(* CoDeSys 2.3.9.36 project: KVR_Mast.bak.pro *)
(* Version: 01 *)
(* Author: JB *)
(* Libraries: ifm_CR0401\ifm_CR0401_V030100.lib*30.7.20 10:49:34, ifm_RAWCan\ifm_RAWCan_NT_V020004.lib*27.10.21 18:23:48, ifm_CANopen\ifm_CANopen_NT_V020004.lib*27.10.21 18:23:48, ifm_CANopen\3S_CanDrv.lib*27.10.21 18:23:48, ifm_CANopen\3S_CANopenManager.lib*27.10.21 18:23:48, Util.lib 6.11.07 15:39:24, standard.lib 4.10.05 12:14:46, SysLibCallback.lib 26.9.08 17:43:52 *)

(* PLC configuration (modules and I/O channels)
Configuration [LocalConfiguration] node 0, in %IB0 out %QB0 {IFM_PARAM_WORD_TIME = 0}
Input/Output [LocalInputOutput] node 1, in %IB0 out %QB0
IN00 AT %IB0 [ChInputBool] Input 00 Bit
IN01 AT %IB1 [ChInputBool] Input 01 Bit
IN02 AT %IB2 [ChInputBool] Input 02 Bit
IN03 AT %IB3 [ChInputBool] Input 03 Bit
IN04 AT %IB4 [ChInputBool] Input 04 Bit
IN05 AT %IB5 [ChInputBool] Input 05 Bit
IN06 AT %IB6 [ChInputBool] Input 06 Bit
IN07 AT %IB7 [ChInputBool] Input 07 Bit
IN08 AT %IB8 [ChInputBool] Input 08 Bit
IN09 AT %IB9 [ChInputBool] Input 09 Bit
IN10 AT %IB10 [ChInputBool] Input 10 Bit
IN11 AT %IB11 [ChInputBool] Input 11 Bit
OUT00 AT %QB0 [ChOutputBool] Output 00 Bit
OUT01 AT %QB1 [ChOutputBool] Output 01 Bit
OUT02 AT %QB2 [ChOutputBool] Output 02 Bit
OUT03 AT %QB3 [ChOutputBool] Output 03 Bit
OUT04 AT %QB4 [ChOutputBool] Output 04 Bit
OUT05 AT %QB5 [ChOutputBool] Output 05 Bit
OUT06 AT %QB6 [ChOutputBool] Output 06 Bit
OUT07 AT %QB7 [ChOutputBool] Output 07 Bit
System Inputs [LocalSystemInputs] node 2, in %IB12 out %QB8
  SUPPLY_VOLTAGE_VBBS AT %IW6 [ChInputWord] Supply voltage VBBS
  SUPPLY_VOLTAGE_VU AT %IW7 [ChInputWord] Supply voltage VU
  SUPPLY_VOLTAGE_VBB1 AT %IW8 [ChInputWord] Supply voltage VBB1
  SUPPLY_VOLTAGE_VBB2 AT %IW9 [ChInputWord] Supply voltage VBB2
  TEMPERATURE AT %IW10 [ChInputInt] Temperature
J1939 Interface [CAN_J1939] node 1, in %IB44 out %QB16
J1939 Interface [CAN_J1939] node 1, in %IB44 out %QB16
*)

(* Global variable list: Global_Constants *)
VAR_GLOBAL CONSTANT

	MAX_CTRLINDEX: BYTE := 0;

	SIMULATIONSMODUS: BOOL := FALSE;

	(* Flag positions for variable FlagsECU2PC *)
	ECU2PC_AllowRemote: INT := 3;
	ECU2PC_EmergencyStop: INT := 4;
	ECU2PC_RemoteAckn: INT := 6;
	ECU2PC_MainSwitch: INT := 7;

	(* Flag positions for variable FlagsPC2ECU *)
	PC2ECU_Remote: INT := 0;
	PC2ECU_BlackOut: INT := 1;
	PC2ECU_ResetMotorActiveTime: INT := 3;

	(* Flag positions for variables Mast[x].FlagsECU2PC *)
	ECU2PC_TopPosition: INT := 0;
	ECU2PC_BottomPosition: INT := 1;
	ECU2PC_MovingUp: INT := 2;
	ECU2PC_MovingDown: INT := 3;
	ECU2PC_LocalUp: INT := 4;
	ECU2PC_LocalDown: INT := 5;
	ECU2PC_LimitSwitch4m: INT := 7;
	ECU2PC_LimitSwitchBottom: INT := 8;
	ECU2PC_NotReadyToSwitchOn: INT := 9;
	ECU2PC_ParkPosition: INT := 10;
	ECU2PC_MontagePos: INT := 11;

	(* Flag positions for variables Mast[x].FlagsPC2ECU *)
	PC2ECU_MoveUp: INT := 0;
	PC2ECU_MoveDown: INT := 1;
	PC2ECU_SlowSpeed: INT := 2;

	(* Flag positions for variable Mast[x].ErrorECU2PC *)
	ECU2PC_ErrorFU: INT 					:= 0;
	ECU2PC_ErrorCanTimeout: INT 			:= 1;
	ECU2PC_ErrorFUPos: INT 					:= 6;
	ECU2PC_ErrorEndschalterUnten1: INT 		:= 7;
	ECU2PC_ErrorEndschalterUnten2: INT 		:= 8;
	ECU2PC_ErrorCurrentLimit: INT			:= 9;
	ECU2PC_ErrorSetMastHeight: INT			:= 10;

	QSCMD_NOP: BYTE				:= 0;
	QSCMD_CLEAR_ERROR: BYTE		:= 1;
	QSCMD_QUICK_STOP: BYTE		:= 113;
	QSCMD_HALT: BYTE			:= 114;
	QSCMD_VELOCITY_MODE: BYTE	:= 117; (* QSData0 = desired velocity *)
	QSCMD_ABS_POS_MODE: BYTE	:= 118; (* QSData0 = desired velocity, QSData1 = desired position *)

	(* Flag positions for FU statusword *)
	STAT_ENABLED: INT			:= 0;
	STAT_ERROR: INT				:= 1;
	STAT_WARNING: INT			:= 2;
	STAT_MOVING: INT			:= 3;
	STAT_REACHED: INT			:= 4;
	STAT_LIMIT: INT				:= 5;
	STAT_STOP_OR_HALT: INT		:= 11;

	FU1_POS_TO_MM: REAL 		:= 3.2573E-004;

	CAN_CHANNEL_HOST: BYTE 		:= 2;
	CAN_CHANNEL_LOCAL: BYTE 	:= 1;

	FU1_NODE_ID: BYTE			:= 127;

END_VAR

(* Global variable list: Global_Variables *)
VAR_GLOBAL

	BlinkSlow: BOOL;

	MasterPresent: BOOL;

	inputs: TYPE_INPUTS;
	outputs: TYPE_OUTPUTS;

	canNodeFU1Present: BOOL;

	tasteAuf: BOOL;
	tasteAb: BOOL;

	FlagsECU2PC: WORD			{parameter list=proc_vars_ecu [name=FlagsECU2PC 					index=16#3000 subindex=1 accessright="read only"] };
	FlagsPC2ECU: WORD			{parameter list=proc_vars_ecu [name=FlagsPC2ECU 					index=16#3000 subindex=2 accessright="write only"] };
	Windspeed: BYTE				{parameter list=proc_vars_ecu [name=Windspeed	 					index=16#3000 subindex=3 accessright="read only"] };
	CabinetTemperature: SINT	{parameter list=proc_vars_ecu [name=Temperature	 					index=16#3000 subindex=4 accessright="read only"] };
	ExtTemperature: SINT		{parameter list=proc_vars_ecu [name=ExtTemperature	 				index=16#3000 subindex=5 accessright="read only"] };
	IntVoltage: WORD			{parameter list=proc_vars_ecu [name=IntVoltage		 				index=16#3000 subindex=6 accessright="read only"] };

	Mast1Height: WORD			{parameter list=proc_vars_mast1 [name=Mast1Height 					index=16#3001 subindex=1 accessright="read only"] };
	Mast1FlagsECU2PC: WORD		{parameter list=proc_vars_mast1 [name=Mast1FlagsECU2PC 				index=16#3003 subindex=1 accessright="read only"] };
	Mast1FlagsPC2ECU: WORD		{parameter list=proc_vars_mast1 [name=Mast1FlagsPC2ECU 				index=16#3004 subindex=1 accessright="write only"] };
	Mast1Current: DINT			{parameter list=proc_vars_mast1 [name=Mast1Current 					index=16#3006 subindex=1 accessright="read only"] };
	Mast1ErrorECU2PC: WORD		{parameter list=proc_vars_mast1 [name=Mast1ErrorECU2PC				index=16#300D subindex=1 accessright="read only"] };
	Mast1FUErrorCode: WORD		{parameter list=proc_vars_mast1 [name=Mast1FUErrorCode				index=16#3010 subindex=1 accessright="read only"] };
	Mast1Speed: DINT			{parameter list=proc_vars_mast1 [name=Mast1Speed					index=16#3013 subindex=1 accessright="read only"] };

	(*
	Mast1TempPcbPower: WORD		{parameter list=proc_vars_mast1 [name=Mast1TempPcbPower				index=16#300A subindex=1 accessright="read only"] };
	Mast1TempPcbController: WORD{parameter list=proc_vars_mast1 [name=Mast1TempPcbController		index=16#300B subindex=1 accessright="read only"] };
	Mast1TempPcbAmplifier: WORD	{parameter list=proc_vars_mast1 [name=Mast1TempPcbAmplifier			index=16#300F subindex=1 accessright="read only"] };
	*)

	Mast1SetEncoderPW: DWORD	{parameter list=Parameters 		[name=Mast1SetEncoderPW				index=16#2014 subindex=1 accessright="read-write"] };

	Version: BYTE				{parameter list=version_info 	[name=Version						index=16#3020 subindex=1 accessright="read only"] };
	VersionDate: DWORD			{parameter list=version_info 	[name=VersionDate					index=16#3020 subindex=2 accessright="read only"] };

	Mast1MotorActiveTimeSeconds2: DWORD {parameter list=proc_vars_mast1 [name=Mast1MotorActiveTimeSeconds2 index=16#3014 subindex=1 accessright="read only"] };

	FU1_Current_Sim: DINT;

END_VAR

(* Global variable list: Parameters *)
VAR_GLOBAL RETAIN
	SettingsPW: DWORD := 0	 					{parameter list=Parameters [name=SettingsPW					 	index=16#2000 subindex=12 accessright="read-write"] };
	Mast1TopPosition: WORD := 9000 				{parameter list=Parameters [name=Mast1TopPosition 				index=16#2006 subindex=1 accessright="read-write"] };
	Mast1BottomPosition: WORD := 1675			{parameter list=Parameters [name=Mast1BottomPosition			index=16#2007 subindex=1 accessright="read-write"] };
	Mast1VelocityNormal: INT := 2500			{parameter list=Parameters [name=Mast1VelocityNormal			index=16#200A subindex=1 accessright="read-write"] };
	Mast1VelocityBottom: INT := 500				{parameter list=Parameters [name=Mast1VelocityBottom			index=16#200C subindex=1 accessright="read-write"] };
	Mast1BottomPositionOffset: WORD := 130		{parameter list=Parameters [name=Mast1BottomPositionOffset		index=16#200D subindex=1 accessright="read-write"] };
	Mast1CurrentLimitBottom: INT := 30			{parameter list=Parameters [name=Mast1CurrentLimitBottom		index=16#200E subindex=1 accessright="read-write"] };
	Mast1BottomLimitSwitchWindow: WORD := 100	{parameter list=Parameters [name=Mast1BottomLimitSwitchWindow	index=16#200F subindex=1 accessright="read-write"] };
	Mast1MontagePos: WORD := 2000 				{parameter list=Parameters [name=Mast1MontagePos 				index=16#2010 subindex=1 accessright="read-write"] };
	Mast1MotorActiveTimeSeconds: DWORD := 0		{parameter list=Parameters [name=Mast1MotorActiveTimeSeconds	index=16#2013 subindex=1 accessright="read-write"] };
	Mast1CurrentLimit: INT := 40				{parameter list=Parameters [name=Mast1CurrentLimit				index=16#2018 subindex=1 accessright="read-write"] };
	Mast1TopSettlingOffset: INT := 40			{parameter list=Parameters [name=Mast1TopSettlingOffset			index=16#2019 subindex=1 accessright="read-write"] };
END_VAR

(* Data type *)
TYPE TYPE_INPUTS :
	STRUCT
		TasteAusfahren: BOOL;
		TasteEinfahren: BOOL;
		TastePoweredByGenerator: BOOL;
		EndschalterNotantrieb: BOOL;
		EndschalterEingefahren: BOOL;
		EndschalterAufgerichtet: BOOL;
	END_STRUCT
END_TYPE

(* Data type *)
TYPE TYPE_OUTPUTS :
	STRUCT
		LEDAusgefahren: BOOL;
		LEDEingefahren: BOOL;
		LEDMontagePos: BOOL;
		RelaisMotorLeistung: BOOL;
		SchuetzGrundlast: BOOL;
	END_STRUCT
END_TYPE

(* POU PLC_PRG, FBD *)
PROGRAM PLC_PRG
VAR
	Init1: BOOL:=TRUE;
	CycleTime:DWORD;
	MaxCycleTime:DWORD;
	ResetMax:BOOL;
END_VAR
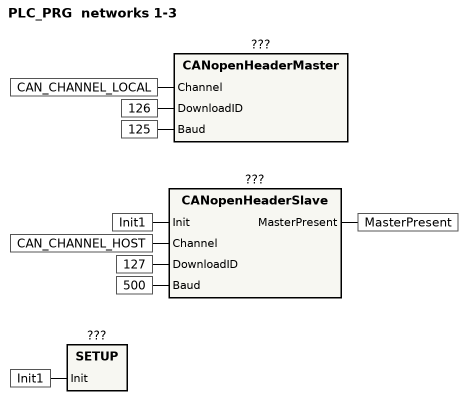
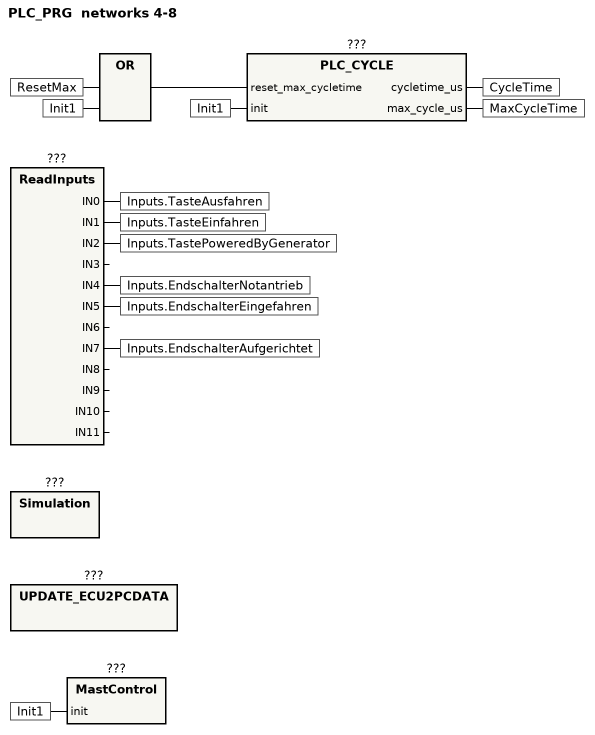
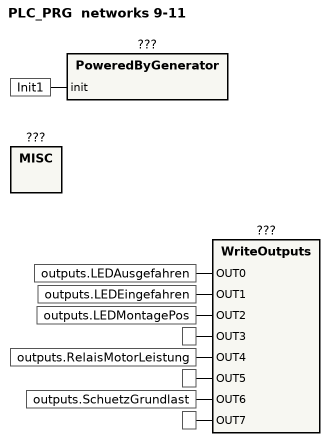
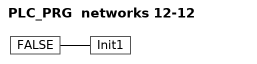
_FBD_ (* Function Block Diagram *)
NETWORK 1 (* CAN Master auf CAN1 initialisieren (Schnittstelle zu FU) *)
	???:CANopenHeaderMaster(Channel: CAN_CHANNEL_LOCAL, DownloadID: 126, Baud: 125)
NETWORK 2 (* CAN Slave auf CAN2 initialisieren (Schnittstelle zu PC) *)
	???:CANopenHeaderSlave(Init: Init1, Channel: CAN_CHANNEL_HOST, DownloadID: 127, Baud: 500) => MasterPresent
NETWORK 3
	???:SETUP(Init: Init1)
NETWORK 4
	???:PLC_CYCLE(reset_max_cycletime: OR(ResetMax, Init1), init: Init1, max_cycle_us => MaxCycleTime) => CycleTime
NETWORK 5
	???:ReadInputs(IN1 => Inputs.TasteEinfahren, IN2 => Inputs.TastePoweredByGenerator, IN4 => Inputs.EndschalterNotantrieb, IN5 => Inputs.EndschalterEingefahren, IN7 => Inputs.EndschalterAufgerichtet) => Inputs.TasteAusfahren
NETWORK 6
	???:Simulation()
NETWORK 7
	???:UPDATE_ECU2PCDATA()
NETWORK 8
	NOT ???:MastControl(init: Init1)
NETWORK 9
	???:PoweredByGenerator(init: Init1)
NETWORK 10
	???:MISC()
NETWORK 11
	???:WriteOutputs(OUT0: outputs.LEDAusgefahren, OUT1: outputs.LEDEingefahren, OUT2: outputs.LEDMontagePos, OUT3: , OUT4: outputs.RelaisMotorLeistung, OUT5: , OUT6: outputs.SchuetzGrundlast, OUT7: )
NETWORK 12 (* last line *)
	FALSE => Init1
_END_FBD_
(* the same logic as Structured Text *)
(* Network 1: see the listing above *)
(* Network 2: see the listing above *)
(* Network 3: see the listing above *)
(* Network 4: see the listing above *)
(* Network 5: see the listing above *)
(* Network 6: see the listing above *)
(* Network 7: see the listing above *)
(* Network 8: see the listing above *)
(* Network 9: see the listing above *)
(* Network 10: see the listing above *)
(* Network 11: see the listing above *)
(* Network 12 *)
Init1 := FALSE;
END_PROGRAM

(* POU CANopen/CANopenHeaderMaster, FBD *)
PROGRAM CANopenHeaderMaster
VAR_INPUT
	Channel: BYTE;
	DownloadID: BYTE;
	Baud: WORD;
END_VAR
VAR
	(*CAN settings*)
	SettingsCAN: CAN_SETTING_ST;

	(*Set CANopen state*)
	SetCanOpenState: CANOPEN_SETSTATE;
	SetState:BOOL:=TRUE;

	(*Handling CANopen status*)
	HandlingCANopen: CANopen_HANDLING_ST;
	Baudrate: DWORD;
	MasterState: BYTE;
	GuardError: BOOL;
	ErrorNodeList: ARRAY[0..MAXGUARDERR] OF BYTE;
	CanState: BYTE;
	Nodestate: BYTE;
	LastNodeState: BYTE;

	(*Emergency handling*)
	CanEmcy: CAN_EMCY;
	RestEmcyList: BOOL;
	EMCY_MSG_Count: DWORD; (* No of EMCY messages  Leaving errors are count too *)
	EmcyStruct: ARRAY[0..10] OF tT_EMCY;

	(*Handling CAN status*)
	StatusCan: CAN_Status_and_Errors;
	ResetCanFlags: BOOL;
	BusLoad: BYTE;
	BusOff: BOOL;
	RxOverflow: BOOL;
	RxWarning: BOOL;
	TxOverflow: BOOL;
	TxWarning: BOOL;

	GetstateSlave1: CANopen_GetStateSlave;

END_VAR
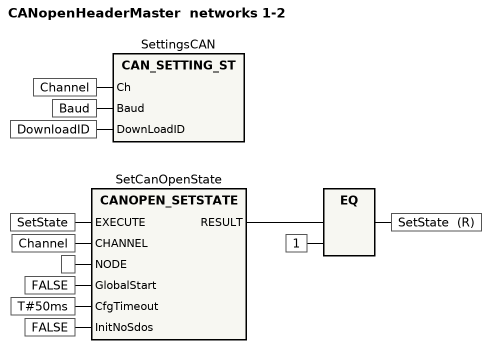
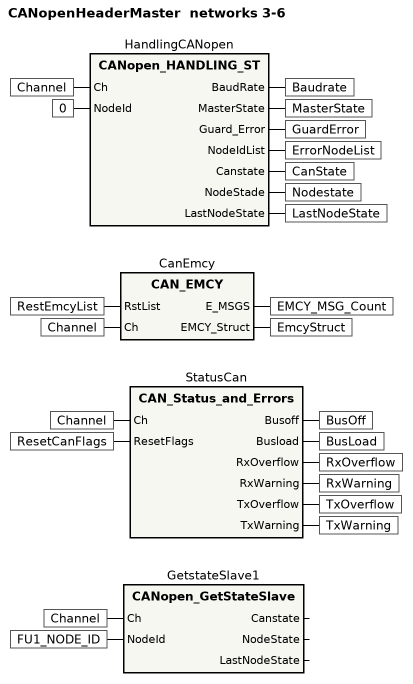
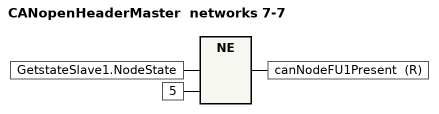
_FBD_ (* Function Block Diagram *)
NETWORK 1 (* Basic functions for the CAN / CANopen functionality *)
	SettingsCAN:CAN_SETTING_ST(Ch: Channel, Baud: Baud, DownLoadID: DownloadID)
NETWORK 2 (* Set CANopen status *)
	EQ(SetCanOpenState:CANOPEN_SETSTATE(EXECUTE: SetState, CHANNEL: Channel, NODE: , GlobalStart: FALSE, CfgTimeout: T#50ms, InitNoSdos: FALSE), 1) => R SetState
NETWORK 3 (* CANopen Master and heartbeat handling *)
	HandlingCANopen:CANopen_HANDLING_ST(Ch: Channel, NodeId: 0, MasterState => MasterState, Guard_Error => GuardError, NodeIdList => ErrorNodeList, Canstate => CanState, NodeStade => Nodestate, LastNodeState => LastNodeState) => Baudrate
NETWORK 4 (* CANopen Emergency Handling for 11 emergency messages *)
	CanEmcy:CAN_EMCY(RstList: RestEmcyList, Ch: Channel, EMCY_Struct => EmcyStruct) => EMCY_MSG_Count
NETWORK 5 (* Get the CAN Status and CAN Errors *)
	StatusCan:CAN_Status_and_Errors(Ch: Channel, ResetFlags: ResetCanFlags, Busload => BusLoad, RxOverflow => RxOverflow, RxWarning => RxWarning, TxOverflow => TxOverflow, TxWarning => TxWarning) => BusOff
NETWORK 6
	GetstateSlave1:CANopen_GetStateSlave(Ch: Channel, NodeId: FU1_NODE_ID)
NETWORK 7
	NE(GetstateSlave1.NodeState, 5) => R canNodeFU1Present
_END_FBD_
(* the same logic as Structured Text *)
(* Network 1 *)
SettingsCAN(Ch := Channel, Baud := Baud, DownLoadID := DownloadID);
(* Network 2: see the listing above *)
(* Network 3 *)
HandlingCANopen(Ch := Channel, NodeId := 0);
MasterState := HandlingCANopen.MasterState;
GuardError := HandlingCANopen.Guard_Error;
ErrorNodeList := HandlingCANopen.NodeIdList;
CanState := HandlingCANopen.Canstate;
Nodestate := HandlingCANopen.NodeStade;
LastNodeState := HandlingCANopen.LastNodeState;
Baudrate := HandlingCANopen.BaudRate;
(* Network 4 *)
CanEmcy(RstList := RestEmcyList, Ch := Channel);
EmcyStruct := CanEmcy.EMCY_Struct;
EMCY_MSG_Count := CanEmcy.E_MSGS;
(* Network 5 *)
StatusCan(Ch := Channel, ResetFlags := ResetCanFlags);
BusLoad := StatusCan.Busload;
RxOverflow := StatusCan.RxOverflow;
RxWarning := StatusCan.RxWarning;
TxOverflow := StatusCan.TxOverflow;
TxWarning := StatusCan.TxWarning;
BusOff := StatusCan.Busoff;
(* Network 6 *)
GetstateSlave1(Ch := Channel, NodeId := FU1_NODE_ID);
(* Network 7 *)
IF GetstateSlave1.NodeState <> 5 THEN canNodeFU1Present := FALSE; END_IF;
END_PROGRAM

(* POU CANopen/CAN_SETTING_ST, ST *)
FUNCTION_BLOCK CAN_SETTING_ST
(* Basic functions for the CAN / CANopen functionality *)
VAR

	CAN_SETDOWNLOADID_: CAN_SETDOWNLOADID;
	CAN_ENABLE_: CAN_ENABLE;
	CANOPEN_ENABLE_: CANOPEN_ENABLE;

	CANOPEN_SETSTATE_: CANOPEN_SETSTATE;
END_VAR
VAR_INPUT
	Ch: BYTE;
	Baud:WORD;
	DownLoadID:BYTE;
END_VAR
CAN_SETDOWNLOADID_(EXECUTE:=TRUE , CHANNEL:=Ch , DOWNLOAD_ID:=DownLoadID , RESULT=> );
CAN_ENABLE_(ENABLE:=TRUE , CHANNEL:=Ch , BAUDRATE:=Baud , RESULT=> );
CANOPEN_ENABLE_(ENABLE:=TRUE , CHANNEL:=Ch , Baudrate:=Baud , RESULT=> );
END_FUNCTION_BLOCK

(* POU CANopen/CANopen_HANDLING_ST, ST *)
FUNCTION_BLOCK CANopen_HANDLING_ST
(* CANopen Master and heartbeat handling *)
VAR
	CANOPEN_GETSTATE_: CANOPEN_GETSTATE;
	Execute_Getstate: BOOL := TRUE;
	CANOPEN_GETGUARDHBERRLIST_: CANOPEN_GETGUARDHBERRLIST;
	Execute_Guardlst: BOOL := TRUE;
	ResetErrorList: BOOL;
	PlcNodeId: BYTE;
	i: INT;
	GuardErrorCnt: WORD;
END_VAR
VAR_INPUT
	Ch: BYTE;
	NodeId: BYTE;
END_VAR
VAR_OUTPUT
	BaudRate: DWORD;
	MasterState: BYTE;
	Guard_Error: BOOL;
	NodeIdList: ARRAY[0..MAXGUARDERR] OF BYTE;
	Canstate: BYTE;
	NodeStade: BYTE;
	LastNodeState: BYTE;
END_VAR
(* ^^^^ Get the current state of the CANopen master ^^^^ *)
CANOPEN_GETSTATE_(
	EXECUTE:=Execute_Getstate ,
	CHANNEL:=Ch ,
	NODE:=NodeId ,
	MASTERSTATE=>MasterState ,
	PLCNODEID=>PlcNodeId ,
	PLCBAUDRATE=>BaudRate ,
	PLCVERSION=>,
	CANSTATE=>Canstate ,
	NODESTATE=>NodeStade ,
	LASTNODESTATE=>LastNodeState ,
	RESULT=> );

(* Values are valid now, function call can be stopped *)
IF CANOPEN_GETSTATE_.RESULT= 1 THEN
	Execute_Getstate:=FALSE;
END_IF

(* Function is passive, execute again *)
IF CANOPEN_GETSTATE_.RESULT= 0 THEN
	Execute_Getstate:=TRUE;
END_IF

(* ^^^^^ Get heartbeaterror or nodeguarding error ^^^^ *)
CANOPEN_GETGUARDHBERRLIST_(
	EXECUTE:=Execute_Guardlst ,
	CHANNEL:=Ch ,
	ResetList:=ResetErrorList ,
	N_NODES=>GuardErrorCnt,
	NODEID=>NodeIdList ,
	RESULT=> );

(* Values are valid now, function call can be stopped *)
IF CANOPEN_GETGUARDHBERRLIST_.RESULT= 1 THEN
	Execute_Guardlst:= FALSE;
END_IF

(* Function is passive, execute again *)
IF CANOPEN_GETGUARDHBERRLIST_.RESULT= 0 THEN
	Execute_Guardlst:= TRUE;
END_IF

(* An heartbeaterror has been appeared *)
IF CANOPEN_GETGUARDHBERRLIST_.N_NODES >0 THEN
	Guard_Error:=TRUE;
ELSE
	Guard_Error:=FALSE;
END_IF;

IF Ch = CAN_CHANNEL_LOCAL THEN

	canNodeFU1Present := TRUE;
	
	FOR i := 0 TO GuardErrorCnt DO
		IF FU1_NODE_ID = NodeIdList[i] THEN
			canNodeFU1Present := FALSE;
		END_IF
	END_FOR

END_IF
END_FUNCTION_BLOCK

(* POU CANopen/CAN_EMCY, FBD *)
FUNCTION_BLOCK CAN_EMCY
VAR_INPUT
	RstList: BOOL;
	Ch: BYTE;
END_VAR
VAR_OUTPUT
	E_MSGS: DWORD;
	EMCY_Struct: ARRAY[0..10] OF tT_EMCY;
END_VAR
VAR
	CANOPEN_GETEMCYMESSAGES_: CANOPEN_GETEMCYMESSAGES;
	Get_EMCY_MSG: BOOL := TRUE;
END_VAR
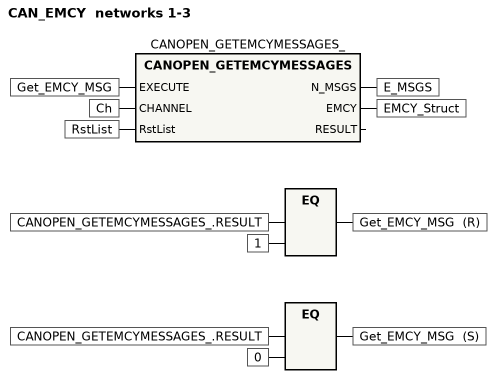
_FBD_ (* Function Block Diagram *)
NETWORK 1
	CANOPEN_GETEMCYMESSAGES_:CANOPEN_GETEMCYMESSAGES(EXECUTE: Get_EMCY_MSG, CHANNEL: Ch, RstList: RstList, EMCY => EMCY_Struct) => E_MSGS
NETWORK 2
	EQ(CANOPEN_GETEMCYMESSAGES_.RESULT, 1) => R Get_EMCY_MSG
NETWORK 3
	EQ(CANOPEN_GETEMCYMESSAGES_.RESULT, 0) => S Get_EMCY_MSG
_END_FBD_
(* the same logic as Structured Text *)
(* Network 1 *)
CANOPEN_GETEMCYMESSAGES_(EXECUTE := Get_EMCY_MSG, CHANNEL := Ch, RstList := RstList);
EMCY_Struct := CANOPEN_GETEMCYMESSAGES_.EMCY;
E_MSGS := CANOPEN_GETEMCYMESSAGES_.N_MSGS;
(* Network 2 *)
IF CANOPEN_GETEMCYMESSAGES_.RESULT = 1 THEN Get_EMCY_MSG := FALSE; END_IF;
(* Network 3 *)
IF CANOPEN_GETEMCYMESSAGES_.RESULT = 0 THEN Get_EMCY_MSG := TRUE; END_IF;
END_FUNCTION_BLOCK

(* POU CANopen/CAN_Status_and_Errors, FBD *)
FUNCTION_BLOCK CAN_Status_and_Errors
(* Get the CAN Status and CAN Errors *)
VAR

	CanStatus:CAN_STATUS;
	GETBUFFERFLAGS: CANOPEN_GETBUFFERFLAGS;

	ExecuteBufferFlags: BOOL:=TRUE;

END_VAR
VAR_INPUT
	Ch: BYTE;

	ResetFlags: BOOL;
END_VAR
VAR_OUTPUT
	Busoff: BOOL;
	Busload: BYTE;
	RxOverflow: BOOL;
	RxWarning: BOOL;
	TxOverflow: BOOL;
	TxWarning: BOOL;
END_VAR
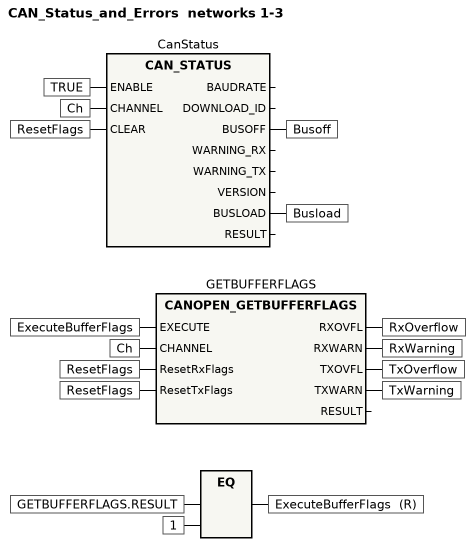
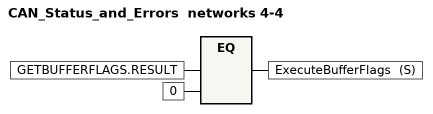
_FBD_ (* Function Block Diagram *)
NETWORK 1 (* Get the CAN Status *)
	CanStatus:CAN_STATUS(ENABLE: TRUE, CHANNEL: Ch, CLEAR: ResetFlags, BUSOFF => Busoff, BUSLOAD => Busload)
NETWORK 2 (* Get Buffer warnings / Reset Buffer Warning *)
	GETBUFFERFLAGS:CANOPEN_GETBUFFERFLAGS(EXECUTE: ExecuteBufferFlags, CHANNEL: Ch, ResetRxFlags: ResetFlags, ResetTxFlags: ResetFlags, RXWARN => RxWarning, TXOVFL => TxOverflow, TXWARN => TxWarning) => RxOverflow
NETWORK 3
	EQ(GETBUFFERFLAGS.RESULT, 1) => R ExecuteBufferFlags
NETWORK 4
	EQ(GETBUFFERFLAGS.RESULT, 0) => S ExecuteBufferFlags
_END_FBD_
(* the same logic as Structured Text *)
(* Network 1: Get the CAN Status *)
CanStatus(ENABLE := TRUE, CHANNEL := Ch, CLEAR := ResetFlags);
Busoff := CanStatus.BUSOFF;
Busload := CanStatus.BUSLOAD;
(* Network 2: Get Buffer warnings / Reset Buffer Warning *)
GETBUFFERFLAGS(EXECUTE := ExecuteBufferFlags, CHANNEL := Ch, ResetRxFlags := ResetFlags, ResetTxFlags := ResetFlags);
RxWarning := GETBUFFERFLAGS.RXWARN;
TxOverflow := GETBUFFERFLAGS.TXOVFL;
TxWarning := GETBUFFERFLAGS.TXWARN;
RxOverflow := GETBUFFERFLAGS.RXOVFL;
(* Network 3 *)
IF GETBUFFERFLAGS.RESULT = 1 THEN ExecuteBufferFlags := FALSE; END_IF;
(* Network 4 *)
IF GETBUFFERFLAGS.RESULT = 0 THEN ExecuteBufferFlags := TRUE; END_IF;
END_FUNCTION_BLOCK

(* POU CANopen/CANopen_GetStateSlave, ST *)
FUNCTION_BLOCK CANopen_GetStateSlave
VAR
	CANOPEN_GETSTATE_: CANOPEN_GETSTATE;
	Execute_Getstate: BOOL := TRUE;
END_VAR
VAR_INPUT
	Ch: BYTE;
	NodeId: BYTE;
END_VAR
VAR_OUTPUT
	Canstate: BYTE;
	NodeState: BYTE;
	LastNodeState: BYTE;
END_VAR
CANOPEN_GETSTATE_(
	EXECUTE:=Execute_Getstate ,
	CHANNEL:=Ch ,
	NODE:=NodeId ,
	MASTERSTATE=>,
	PLCNODEID=> ,
	PLCBAUDRATE=> ,
	PLCVERSION=>,
	CANSTATE=>Canstate ,
	NODESTATE=>NodeState ,
	LASTNODESTATE=>LastNodeState ,
	RESULT=> );

(* Values are valid now, function call can be stopped *)
IF CANOPEN_GETSTATE_.RESULT= 1 THEN
	Execute_Getstate:=FALSE;
END_IF

(* Function is passive, execute again *)
IF CANOPEN_GETSTATE_.RESULT= 0 THEN
	Execute_Getstate:=TRUE;
END_IF
END_FUNCTION_BLOCK

(* POU CANopen/CANopenHeaderSlave, FBD *)
PROGRAM CANopenHeaderSlave
VAR_INPUT
	Init: BOOL;
	Channel: BYTE;
	DownloadID: BYTE;
	Baud: WORD;
END_VAR
VAR_OUTPUT
	MasterPresent: BOOL;
END_VAR
VAR
	(*SettingsCAN*)
	SettingsCAN: CAN_SETTING_ST;

	(*Get status*)
	GetStateSlave: CANOPEN_GETNMTSTATESLAVE;
	SetGetStateSlave: BOOL;
	ResultState: BYTE;
	NodeState: BYTE;

	(*Get CANopen Node ID*)
	GetState: CANOPEN_GETSTATE;
	NodeId: BYTE;

	(*Get Guarding status*)
	GetGuard: CANOPEN_GETGUARDHBSTATSLV;
	GetGuardEx: BOOL;
	ResetGuard: BOOL;

END_VAR
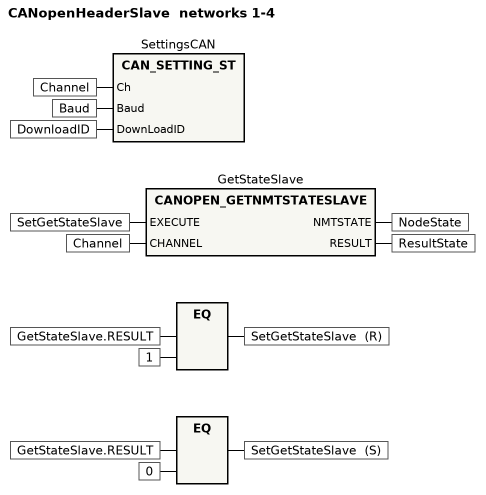
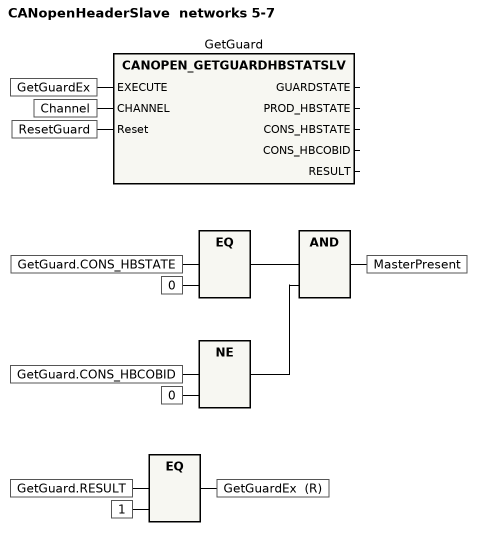
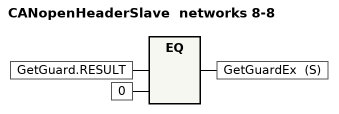
_FBD_ (* Function Block Diagram *)
NETWORK 1 (* Basic functions for the CAN / CANopen functionality *)
	SettingsCAN:CAN_SETTING_ST(Ch: Channel, Baud: Baud, DownLoadID: DownloadID)
NETWORK 2
	GetStateSlave:CANOPEN_GETNMTSTATESLAVE(EXECUTE: SetGetStateSlave, CHANNEL: Channel, RESULT => ResultState) => NodeState
NETWORK 3
	EQ(GetStateSlave.RESULT, 1) => R SetGetStateSlave
NETWORK 4
	EQ(GetStateSlave.RESULT, 0) => S SetGetStateSlave
NETWORK 5
	GetGuard:CANOPEN_GETGUARDHBSTATSLV(EXECUTE: GetGuardEx, CHANNEL: Channel, Reset: ResetGuard)
NETWORK 6
	AND(EQ(GetGuard.CONS_HBSTATE, 0), NE(GetGuard.CONS_HBCOBID, 0)) => MasterPresent
NETWORK 7
	EQ(GetGuard.RESULT, 1) => R GetGuardEx
NETWORK 8
	EQ(GetGuard.RESULT, 0) => S GetGuardEx
_END_FBD_
(* the same logic as Structured Text *)
(* Network 1: Basic functions for the CAN / CANopen functionality *)
SettingsCAN(Ch := Channel, Baud := Baud, DownLoadID := DownloadID);
(* Network 2 *)
GetStateSlave(EXECUTE := SetGetStateSlave, CHANNEL := Channel);
ResultState := GetStateSlave.RESULT;
NodeState := GetStateSlave.NMTSTATE;
(* Network 3 *)
IF GetStateSlave.RESULT = 1 THEN SetGetStateSlave := FALSE; END_IF;
(* Network 4 *)
IF GetStateSlave.RESULT = 0 THEN SetGetStateSlave := TRUE; END_IF;
(* Network 5 *)
GetGuard(EXECUTE := GetGuardEx, CHANNEL := Channel, Reset := ResetGuard);
(* Network 6 *)
MasterPresent := (GetGuard.CONS_HBSTATE = 0) AND (GetGuard.CONS_HBCOBID <> 0);
(* Network 7 *)
IF GetGuard.RESULT = 1 THEN GetGuardEx := FALSE; END_IF;
(* Network 8 *)
IF GetGuard.RESULT = 0 THEN GetGuardEx := TRUE; END_IF;
END_PROGRAM

(* POU Steuerung/SETUP, ST *)
PROGRAM SETUP
VAR_INPUT
	Init: BOOL;
END_VAR
VAR
	getAppInfo: GET_APP_INFO;
END_VAR
IF NOT Init THEN
	RETURN;
END_IF;

Mast1FlagsECU2PC.ECU2PC_ParkPosition := FALSE;

getAppInfo(ENABLE := TRUE);

VersionDate := STRING_TO_DWORD(LEFT(getAppInfo.BUILD_DATE, 8));
Version := STRING_TO_BYTE(LEFT(getAppInfo.VERSION, 3));
END_PROGRAM

(* POU PLC_CYCLE, ST *)
PROGRAM PLC_CYCLE
VAR_INPUT
	reset_max_cycletime: BOOL;
	init: BOOL;
END_VAR
VAR_OUTPUT
	cycletime_us: DWORD;
	max_cycle_us: DWORD;
END_VAR
VAR
	old_cycle: DWORD;
	TIMER_READ_US1: TIMER_READ_US;
	cycle: DWORD;
	nextTS: DWORD;
END_VAR
TIMER_READ_US1(TIME_US=>cycle );
cycletime_us:=cycle-old_cycle;
old_cycle:=cycle;

IF max_cycle_us<cycletime_us AND NOT init THEN
	max_cycle_us:=cycletime_us;
END_IF

IF reset_max_cycletime THEN
	max_cycle_us:=0;
END_IF

IF init THEN
	nextTS := cycle;
END_IF
(* Mehr als 1 Mio Ticks vergangen? *)
(* Zweikomplementarithmetik, d.h. funktioniert auch bei DWORD-Überlauf *)
IF cycle - nextTS > 1000000 THEN
	(* Das nächste Mal wieder nach 1 Mio Ticks (=1 Sekunde) *)
	nextTS := nextTS + 1000000;
	IF FU1_QSCmd <> QSCMD_HALT THEN
		Mast1MotorActiveTimeSeconds := Mast1MotorActiveTimeSeconds + 1;
	END_IF
END_IF
IF FlagsPC2ECU.PC2ECU_ResetMotorActiveTime THEN
	Mast1MotorActiveTimeSeconds := 0;
END_IF
END_PROGRAM

(* POU InputsOutputs/ReadInputs, FBD *)
PROGRAM ReadInputs
VAR
	_input: ARRAY[0..11] OF INPUT;
END_VAR
VAR_OUTPUT
	IN0: BOOL;
	IN1: BOOL;
	IN2: BOOL;
	IN3: BOOL;
	IN4: BOOL;
	IN5: BOOL;
	IN6: BOOL;
	IN7: BOOL;
	IN8: BOOL;
	IN9: BOOL;
	IN10: BOOL;
	IN11: BOOL;
END_VAR
VAR CONSTANT
	ModeInput_Off: BYTE := 0;
	ModeInput_0_10V: BYTE := 3;
	ModeInput_Ratio: BYTE := 6;
	ModeInput_0_20mA: BYTE := 7;
	ModeInput_0_32V: BYTE := 9;
	ModeInput_LowSide: BYTE := 10;
	ModeInput_LowSideNamur: BYTE := 11;
	ModeInput_HighSide: BYTE := 12;
	ModeInput_Resistor: BYTE := 18;
END_VAR
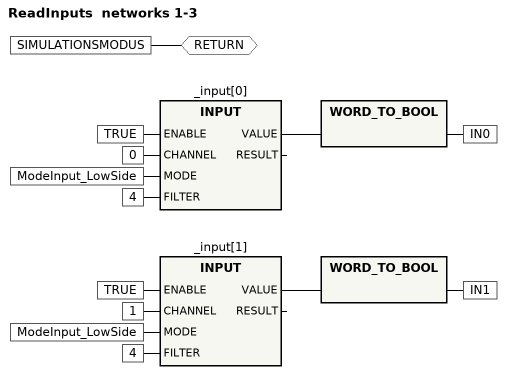
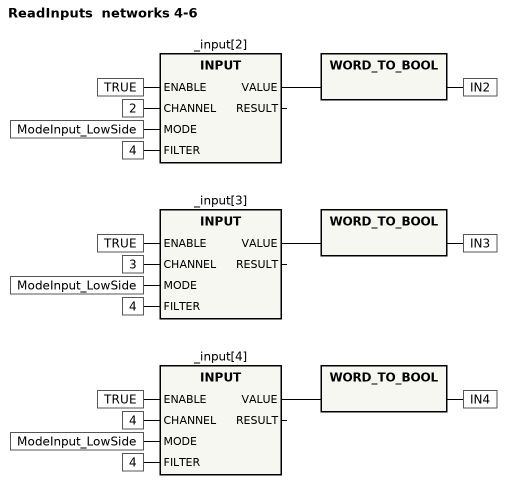
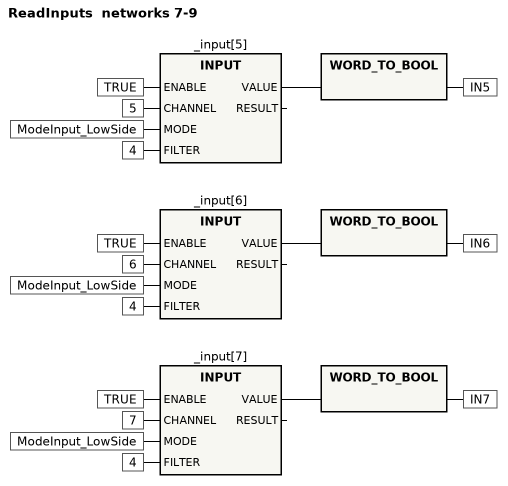
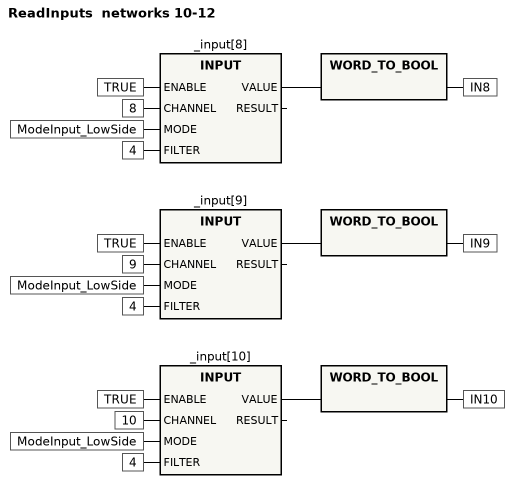
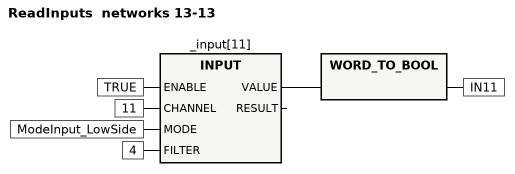
_FBD_ (* Function Block Diagram *)
NETWORK 1
	SIMULATIONSMODUS => <RETURN>
NETWORK 2
	WORD_TO_BOOL(_input[0]:INPUT(ENABLE: TRUE, CHANNEL: 0, MODE: ModeInput_LowSide, FILTER: 4)) => IN0
NETWORK 3
	WORD_TO_BOOL(_input[1]:INPUT(ENABLE: TRUE, CHANNEL: 1, MODE: ModeInput_LowSide, FILTER: 4)) => IN1
NETWORK 4
	WORD_TO_BOOL(_input[2]:INPUT(ENABLE: TRUE, CHANNEL: 2, MODE: ModeInput_LowSide, FILTER: 4)) => IN2
NETWORK 5
	WORD_TO_BOOL(_input[3]:INPUT(ENABLE: TRUE, CHANNEL: 3, MODE: ModeInput_LowSide, FILTER: 4)) => IN3
NETWORK 6
	WORD_TO_BOOL(_input[4]:INPUT(ENABLE: TRUE, CHANNEL: 4, MODE: ModeInput_LowSide, FILTER: 4)) => IN4
NETWORK 7
	WORD_TO_BOOL(_input[5]:INPUT(ENABLE: TRUE, CHANNEL: 5, MODE: ModeInput_LowSide, FILTER: 4)) => IN5
NETWORK 8
	WORD_TO_BOOL(_input[6]:INPUT(ENABLE: TRUE, CHANNEL: 6, MODE: ModeInput_LowSide, FILTER: 4)) => IN6
NETWORK 9
	WORD_TO_BOOL(_input[7]:INPUT(ENABLE: TRUE, CHANNEL: 7, MODE: ModeInput_LowSide, FILTER: 4)) => IN7
NETWORK 10
	WORD_TO_BOOL(_input[8]:INPUT(ENABLE: TRUE, CHANNEL: 8, MODE: ModeInput_LowSide, FILTER: 4)) => IN8
NETWORK 11
	WORD_TO_BOOL(_input[9]:INPUT(ENABLE: TRUE, CHANNEL: 9, MODE: ModeInput_LowSide, FILTER: 4)) => IN9
NETWORK 12
	WORD_TO_BOOL(_input[10]:INPUT(ENABLE: TRUE, CHANNEL: 10, MODE: ModeInput_LowSide, FILTER: 4)) => IN10
NETWORK 13
	WORD_TO_BOOL(_input[11]:INPUT(ENABLE: TRUE, CHANNEL: 11, MODE: ModeInput_LowSide, FILTER: 4)) => IN11
_END_FBD_
(* the same logic as Structured Text *)
(* Network 1 *)
IF SIMULATIONSMODUS THEN RETURN; END_IF;
(* Network 2 *)
_input[0](ENABLE := TRUE, CHANNEL := 0, MODE := ModeInput_LowSide, FILTER := 4);
IN0 := WORD_TO_BOOL(_input[0].VALUE);
(* Network 3 *)
_input[1](ENABLE := TRUE, CHANNEL := 1, MODE := ModeInput_LowSide, FILTER := 4);
IN1 := WORD_TO_BOOL(_input[1].VALUE);
(* Network 4 *)
_input[2](ENABLE := TRUE, CHANNEL := 2, MODE := ModeInput_LowSide, FILTER := 4);
IN2 := WORD_TO_BOOL(_input[2].VALUE);
(* Network 5 *)
_input[3](ENABLE := TRUE, CHANNEL := 3, MODE := ModeInput_LowSide, FILTER := 4);
IN3 := WORD_TO_BOOL(_input[3].VALUE);
(* Network 6 *)
_input[4](ENABLE := TRUE, CHANNEL := 4, MODE := ModeInput_LowSide, FILTER := 4);
IN4 := WORD_TO_BOOL(_input[4].VALUE);
(* Network 7 *)
_input[5](ENABLE := TRUE, CHANNEL := 5, MODE := ModeInput_LowSide, FILTER := 4);
IN5 := WORD_TO_BOOL(_input[5].VALUE);
(* Network 8 *)
_input[6](ENABLE := TRUE, CHANNEL := 6, MODE := ModeInput_LowSide, FILTER := 4);
IN6 := WORD_TO_BOOL(_input[6].VALUE);
(* Network 9 *)
_input[7](ENABLE := TRUE, CHANNEL := 7, MODE := ModeInput_LowSide, FILTER := 4);
IN7 := WORD_TO_BOOL(_input[7].VALUE);
(* Network 10 *)
_input[8](ENABLE := TRUE, CHANNEL := 8, MODE := ModeInput_LowSide, FILTER := 4);
IN8 := WORD_TO_BOOL(_input[8].VALUE);
(* Network 11 *)
_input[9](ENABLE := TRUE, CHANNEL := 9, MODE := ModeInput_LowSide, FILTER := 4);
IN9 := WORD_TO_BOOL(_input[9].VALUE);
(* Network 12 *)
_input[10](ENABLE := TRUE, CHANNEL := 10, MODE := ModeInput_LowSide, FILTER := 4);
IN10 := WORD_TO_BOOL(_input[10].VALUE);
(* Network 13 *)
_input[11](ENABLE := TRUE, CHANNEL := 11, MODE := ModeInput_LowSide, FILTER := 4);
IN11 := WORD_TO_BOOL(_input[11].VALUE);
END_PROGRAM

(* POU Steuerung/Simulation, ST *)
PROGRAM Simulation
VAR
	cnt: WORD;
END_VAR
IF NOT SIMULATIONSMODUS THEN
	RETURN;
END_IF

inputs.EndschalterEingefahren := Mast1Height <= Mast1BottomPosition+2;

IF Mast1Height < Mast1BottomPosition THEN
	Mast1Height := Mast1BottomPosition;
END_IF

FU1_Current_Sim := 0;

IF FU1_QSCmd = QSCMD_ABS_POS_MODE THEN
	IF MastControl.zielposition > Mast1Height THEN
		Mast1Height := Mast1Height + 1;
		FU1_Current_Sim := 10;
	END_IF
	IF MastControl.zielposition < Mast1Height THEN
		Mast1Height := Mast1Height - 1;
		FU1_Current_Sim := 10;
	END_IF
ELSIF FU1_QSCmd = QSCMD_VELOCITY_MODE THEN
	IF cnt > 0 THEN
		cnt := cnt - 1;
	ELSE
		cnt := 10;
		Mast1Height := Mast1Height - 1;
	END_IF
	IF Mast1Height = Mast1BottomPosition THEN
		FU1_Current_Sim := 35;
	ELSE
		FU1_Current_Sim := 10;
	END_IF
END_IF
END_PROGRAM

(* POU Steuerung/MastControl, ST *)
PROGRAM MastControl
VAR_INPUT
	init: BOOL;
END_VAR
VAR
	aufbauen: BOOL;
	abbauen: BOOL;
	zielposition: WORD := 1;
	rtTasteAuf: R_TRIG;
	rtTasteAb: R_TRIG;
	rtTasteReset: R_TRIG;
	rtMastEingefahren: R_TRIG;
	rtSystemEin: R_TRIG;
	resetMasthoehe: BOOL;
	masthoeheReal: REAL;
	FUValue: DWORD;
	SDOWriteOffset: CANOPEN_SDOWRITE;
	SDOData: ARRAY[0..3] OF BYTE;
	TSStart: DWORD;
	tonSystemEin: TON;
	tonKompressor: TON;
	rtResetMasthoehe: R_TRIG;
	statusOffset: BYTE := STATUS_IDLE;
	tofInit: TOF;
	mastPosKorrekt: BOOL := FALSE;
	errorCode71x: BOOL;
	handbetrieb: BOOL := TRUE;
	blnk: BLINK;
	triggerResetMasthoehe: BOOL := FALSE;
	abbauenNullfahrt: BOOL;
	masthoeheSchleichfahrt: WORD;
	masthoeheEndschalter: WORD;
	masthoeheAbsetzen: WORD;
	mastAbsetzen: BOOL := FALSE;
	mastOben: BOOL := FALSE;
	flagTmp: BOOL;
	(* SDOWriteSave: CANOPEN_SDOWRITE; *)
END_VAR
VAR CONSTANT
	_100ms: DWORD := 100000;
	STATUS_IDLE: BYTE := 0;
	STATUS_SETUP_OFFSET: BYTE := 1;
	STATUS_WRITE_OFFSET: BYTE := 2;
	(* STATUS_SETUP_SAVE: BYTE := 3; *)
	(* STATUS_WRITE_SAVE: BYTE := 4; *)
END_VAR
IF NOT SIMULATIONSMODUS THEN
	masthoeheReal := DINT_TO_REAL(FU1_Position) * FU1_POS_TO_MM;
	Mast1Height := REAL_TO_WORD(masthoeheReal);
	Mast1Current := FU1_Current;
ELSE
	Mast1Current := FU1_Current_Sim;
END_IF
Mast1FUErrorCode := FU1_ErrorCode;
Mast1Speed := FU1_Velocity;

(******************* Diverse Timer *******************)
tonSystemEin(IN := TRUE, PT := T#1000ms);
tofInit(IN := init, PT := T#5s);
rtSystemEin(CLK := NOT tofInit.Q);
blnk(ENABLE := TRUE, TIMELOW := T#200ms, TIMEHIGH := T#200ms);

(******************* Initialisierungen *******************)
outputs.RelaisMotorLeistung := FALSE;
FU1_QSCmd := QSCMD_HALT;
masthoeheSchleichfahrt := Mast1BottomPosition + Mast1BottomPositionOffset;
masthoeheEndschalter := Mast1BottomPosition + Mast1BottomLimitSwitchWindow;
masthoeheAbsetzen := Mast1TopPosition - Mast1TopSettlingOffset;
abbauenNullfahrt := FALSE;

(******************* Tasten Flankenerkennung *******************)
rtTasteAuf(CLK := tasteAuf);
rtTasteAb(CLK := tasteAb);
rtTasteReset(CLK := tasteAuf AND tasteAb);

(******************* Flag Mast-Position korrekt falls Endschalter betätigt und Masthöhe plausibel *******************)
(******************* -> Fehlermeldung Masthöhe unterdrücken, keine Nullfahrt notwendig *******************)
IF rtSystemEin.Q THEN
	mastPosKorrekt :=
		inputs.EndschalterEingefahren
		AND Mast1BottomPosition - 2 <= Mast1Height
		AND Mast1Height <= Mast1BottomPosition + 2;
END_IF

(******************* Taste Reset *******************)
IF rtTasteReset.Q THEN
	(* Positionsfehler FU hier nicht zuruecksetzen *)
	flagTmp := Mast1ErrorECU2PC.ECU2PC_ErrorFUPos;
	Mast1ErrorECU2PC := 0;
	Mast1ErrorECU2PC.ECU2PC_ErrorFUPos := flagTmp;
END_IF

(******************* Fehlermeldungen *******************)
Mast1ErrorECU2PC.ECU2PC_ErrorCanTimeout := NOT canNodeFU1Present AND NOT SIMULATIONSMODUS;

(* Auswertung FU Fehlercode *)
(* -710 -> Position unbekannt *)
(* -711 -> Positionswert ungültig *)
errorCode71x := FU1_ErrorCode = -710 OR FU1_ErrorCode = -711;

IF canNodeFU1Present AND tonSystemEin.Q AND FU1_ErrorCode <> 0 THEN
	IF errorCode71x THEN
		IF NOT inputs.EndschalterEingefahren AND NOT mastPosKorrekt THEN
			Mast1ErrorECU2PC.ECU2PC_ErrorFUPos := TRUE;
		END_IF
	ELSE
		Mast1ErrorECU2PC.ECU2PC_ErrorFU := TRUE;
	END_IF
END_IF
IF Mast1Height > masthoeheSchleichfahrt AND inputs.EndschalterEingefahren AND NOT Mast1ErrorECU2PC.ECU2PC_ErrorFUPos AND NOT tofinit.q THEN
	Mast1ErrorECU2PC.ECU2PC_ErrorEndschalterUnten1 := TRUE;
END_IF

(******************* Taste Auf Hand/Auto *******************)
IF rtTasteAuf.Q AND NOT tasteAb THEN
	IF abbauen THEN
		abbauen := FALSE;
	ELSE
		aufbauen := NOT aufbauen;
	END_IF
END_IF
IF NOT tasteAuf AND handbetrieb
 THEN
	aufbauen := FALSE;
END_IF

(******************* Taste Ab Hand/Auto *******************)
IF rtTasteAb.Q AND NOT tasteAuf THEN
	IF aufbauen THEN
		aufbauen := FALSE;
	ELSE
		abbauen := NOT abbauen;
	END_IF
END_IF
IF NOT tasteAuf AND handbetrieb THEN
	abbauen := tasteAb;
END_IF

(******************* Fehler *******************)
IF ABS(Mast1Current) > Mast1CurrentLimit THEN
	Mast1ErrorECU2PC.ECU2PC_ErrorCurrentLimit := TRUE;
END_IF

(******************* Not-Aus / System Aus / Fehler *******************)
IF NOT tonSystemEin.Q OR Mast1ErrorECU2PC <> 0 THEN
	aufbauen := FALSE;
    IF abbauen AND (Mast1ErrorECU2PC.ECU2PC_ErrorFUPos OR NOT mastPosKorrekt) THEN
		abbauenNullfahrt := TRUE;
	END_IF
	abbauen := FALSE;
END_IF

(******************* Zielposition *******************)
IF aufbauen THEN
	IF inputs.EndschalterAufgerichtet THEN
		zielposition := Mast1TopPosition;
	ELSE
		zielposition := Mast1MontagePos;
	END_IF
END_IF
IF abbauen THEN
	zielposition := Mast1BottomPosition;
END_IF

(******************* Aufbauen beendet? *******************)
IF aufbauen AND Mast1Height >= zielposition THEN
	aufbauen := FALSE;
	IF Mast1Height >= Mast1TopPosition THEN
		mastAbsetzen := TRUE;
	END_IF
END_IF

(******************* Abbauen beendet? *******************)
IF abbauen AND Mast1Height <= Mast1BottomPosition THEN
	abbauen := FALSE;
END_IF

(******************* Mast absetzen beendet? *******************)
IF mastAbsetzen AND Mast1Height <= masthoeheAbsetzen THEN
	mastAbsetzen := FALSE;
	mastOben := TRUE;
END_IF

(******************* Fahrbefehle Aufbauen *******************)
IF aufbauen THEN
	mastOben := FALSE;
	FU1_QSData0 := Mast1VelocityNormal;
	FU1_QSData1 := REAL_TO_DINT(WORD_TO_REAL(zielposition)/FU1_POS_TO_MM);
	FU1_QSCmd := QSCMD_ABS_POS_MODE;
END_IF

(******************* Fahrbefehle Abbauen *******************)
IF abbauen THEN
	mastOben := FALSE;
	IF Mast1Height > masthoeheSchleichfahrt THEN
		(* Oberhalb Position Schleichfahrt: Normale Geschwindigkeit *)
		IF NOT resetMasthoehe THEN
			FU1_QSData0 := Mast1VelocityNormal;
			FU1_QSData1 := REAL_TO_DINT(WORD_TO_REAL(masthoeheSchleichfahrt)/FU1_POS_TO_MM);
			FU1_QSCmd := QSCMD_ABS_POS_MODE;
		END_IF
	ELSIF Mast1Height > Mast1BottomPosition THEN
		(* Unterhalb Position Schleichfahrt: Langsame Geschwindigkeit *)
		IF ABS(Mast1Current) > Mast1CurrentLimitBottom THEN
			Mast1ErrorECU2PC.ECU2PC_ErrorCurrentLimit := TRUE;
		ELSIF NOT inputs.EndschalterEingefahren THEN
			Mast1ErrorECU2PC.ECU2PC_ErrorEndschalterUnten2 := TRUE;
		ELSIF NOT resetMasthoehe THEN
			FU1_QSData0 := Mast1VelocityBottom;
	        FU1_QSData1 := REAL_TO_DINT(WORD_TO_REAL(Mast1BottomPosition)/FU1_POS_TO_MM);
			FU1_QSCmd := QSCMD_ABS_POS_MODE;
		END_IF
	END_IF
END_IF

(******************* Fahrbefehle Abbauen Nullfahrt *******************)
IF abbauenNullfahrt THEN
	mastOben := FALSE;
	IF ABS(Mast1Current) > Mast1CurrentLimitBottom THEN
		Mast1ErrorECU2PC.ECU2PC_ErrorCurrentLimit := TRUE;
	ELSIF NOT resetMasthoehe THEN
		IF NOT mastPosKorrekt THEN
			(* Velocity mode: pos = auffahren, neg = einfahren *)
			FU1_QSData0 := -Mast1VelocityBottom;
			FU1_QSCmd := QSCMD_VELOCITY_MODE;
		END_IF
	END_IF
END_IF

(******************* Fahrbefehle Mast auf Riegel absetzen *******************)
IF mastAbsetzen THEN
	mastOben := FALSE;
	FU1_QSData0 := Mast1VelocityNormal;
	FU1_QSData1 := REAL_TO_DINT(WORD_TO_REAL(masthoeheAbsetzen)/FU1_POS_TO_MM);
	FU1_QSCmd := QSCMD_ABS_POS_MODE;
END_IF

(******************* FU-Fehler zurücksetzen *******************)
IF rtTasteReset.Q OR errorCode71x OR NOT tonSystemEin.Q AND blnk.OUT THEN
	FU1_QSCmd := QSCMD_CLEAR_ERROR;
	IF NOT errorCode71x THEN
    	aufbauen := FALSE;
    	abbauen := FALSE;
	END_IF
END_IF

(******************* K1 Versorgung Motor *******************)
outputs.RelaisMotorLeistung := TRUE;

(******************* Masthöhe in FU schreiben bei Schleichfahrt auf Endschalter *******************)
rtMastEingefahren(CLK := inputs.EndschalterEingefahren);
IF NOT resetMasthoehe
	AND rtMastEingefahren.Q
	AND (Mast1BottomPosition < Mast1Height AND Mast1Height < masthoeheSchleichfahrt OR abbauenNullfahrt OR tofInit.Q)
	(* Reset nach Einschalten verhindern *)
	(* AND NOT tofInit.Q *)
THEN
	resetMasthoehe := TRUE;
END_IF


(******************* Masthöhe in FU schreiben falls von Host angefordert *******************)
rtResetMasthoehe(CLK := Mast1SetEncoderPW = 333777333);
IF rtResetMasthoehe.Q THEN
	IF NOT resetMasthoehe
		AND FU1_QSCmd = QSCMD_HALT
		AND inputs.EndschalterEingefahren
	THEN
		resetMasthoehe := TRUE;
	ELSE
		Mast1SetEncoderPW := 101;
	END_IF
END_IF

(******************* Schrittkette Masthöhe in FU schreiben *******************)
CASE statusOffset OF
	STATUS_IDLE:
		IF resetMasthoehe THEN
			statusOffset := STATUS_SETUP_OFFSET;
		END_IF

	STATUS_SETUP_OFFSET:
		(* Masthöhe für Endschalter-Position in FU schreiben *)
		FUValue := REAL_TO_DWORD(masthoeheEndschalter/FU1_POS_TO_MM);
		DWORD_TO_BYTES(
			dw := FUValue,
			ll => SDOData[0],
			ml => SDOData[1],
			mh => SDOData[2],
			hh => SDOData[3]);
		TSStart := PLC_CYCLE.cycle;
		statusOffset := STATUS_WRITE_OFFSET;

	STATUS_WRITE_OFFSET:
		IF PLC_CYCLE.cycle - TSStart > 2*_100ms THEN
			(* 200ms warten, dann prüfen ob Masthöhe unterer Position entspricht *)
			resetMasthoehe := FALSE;
			(* Fehlermeldung Mastposition zurücksetzen *)
			Mast1ErrorECU2PC.ECU2PC_ErrorFUPos := FALSE;
			IF Mast1Height = masthoeheEndschalter THEN
				mastPosKorrekt := TRUE;
				(* statusOffset := STATUS_SETUP_SAVE; 'save' nicht mehr an FU schicken *)
				statusOffset := STATUS_IDLE;
			ELSE
				Mast1ErrorECU2PC.ECU2PC_ErrorSetMastHeight := TRUE;
				CASE SDOWriteOffset.RESULT OF
					1: (* FB-Ausführung wurde ohne Fehler beendet, Daten sind gültig *)
						Mast1SetEncoderPW := 102;
					32: (* SDO-Übertragung abgebrochen von Client oder Server *)
						Mast1SetEncoderPW := 103;
					33: (* TIMEOUT ist abgelaufen *)
						Mast1SetEncoderPW := 104;
					242: (* Fehler: Einstellung ist nicht möglich *)
						Mast1SetEncoderPW := 105;
					ELSE
						Mast1SetEncoderPW := 106;
				END_CASE
				statusOffset := STATUS_IDLE;
			END_IF
		END_IF

	(*
	STATUS_SETUP_SAVE:
		(* Parameter permanent in FU speichern *)
		TSStart := PLC_CYCLE.cycle;
		DWORD_TO_BYTES(
			dw := 16#65766173, (* 'save' *)
			ll => SDOData[0],
			ml => SDOData[1],
			mh => SDOData[2],
			hh => SDOData[3]);
		statusOffset := STATUS_WRITE_SAVE;

	STATUS_WRITE_SAVE:
		IF SDOWriteSave.RESULT = 1 OR PLC_CYCLE.cycle - TSStart > 110*_100ms THEN
			CASE SDOWriteSave.RESULT OF
				1: (* FB-Ausführung wurde ohne Fehler beendet, Daten sind gültig *)
					Mast1SetEncoderPW := 0;
					Mast1ErrorECU2PC.ECU2PC_ErrorSetMastHeight := FALSE;
				32: (* SDO-Übertragung abgebrochen von Client oder Server *)
					Mast1SetEncoderPW := 113;
					Mast1ErrorECU2PC.ECU2PC_ErrorSetMastHeight := TRUE;
				33: (* TIMEOUT ist abgelaufen *)
					Mast1SetEncoderPW := 114;
					Mast1ErrorECU2PC.ECU2PC_ErrorSetMastHeight := TRUE;
				242: (* Fehler: Einstellung ist nicht möglich *)
					Mast1SetEncoderPW := 115;
					Mast1ErrorECU2PC.ECU2PC_ErrorSetMastHeight := TRUE;
				ELSE
					Mast1SetEncoderPW := 116;
					Mast1ErrorECU2PC.ECU2PC_ErrorSetMastHeight := TRUE;
			END_CASE
			statusOffset := STATUS_IDLE;
		END_IF
	*)
END_CASE

(******************* SDO-Befehle *******************)

SDOWriteOffset(
	EXECUTE := statusOffset = STATUS_WRITE_OFFSET,
	CHANNEL := CAN_CHANNEL_LOCAL,
	NODE := FU1_NODE_ID,
	IDX := 16#4762,
	SUBIDX := 1,
	LEN := 4,
	DATA := SDOData,
	Timeout := T#100ms,
	RESULT => );

(*
SDOWriteSave(
	EXECUTE := statusOffset = STATUS_WRITE_SAVE,
	CHANNEL := CAN_CHANNEL_LOCAL,
	NODE := FU1_NODE_ID,
	IDX := 16#1010,
	SUBIDX := 6,
	LEN := 4,
	DATA := SDOData,
	Timeout := T#10s,
	RESULT => );
*)
END_PROGRAM

(* POU Misc/DWORD_TO_BYTES, ST *)
PROGRAM DWORD_TO_BYTES
VAR_INPUT
	dw: DWORD;
END_VAR
VAR_OUTPUT
	ll: BYTE;
	ml: BYTE;
	mh: BYTE;
	hh: BYTE;
END_VAR
ll := DWORD_TO_BYTE(dw);
ml := DWORD_TO_BYTE(SHR(dw, 8));
mh := DWORD_TO_BYTE(SHR(dw, 16));
hh := DWORD_TO_BYTE(SHR(dw, 24));
END_PROGRAM

(* POU Steuerung/UPDATE_ECU2PCDATA, ST *)
PROGRAM UPDATE_ECU2PCDATA
FlagsECU2PC.ECU2PC_AllowRemote := TRUE;

FlagsECU2PC.ECU2PC_EmergencyStop := FALSE;

FlagsECU2PC.ECU2PC_RemoteAckn := FALSE;

FlagsECU2PC.ECU2PC_MainSwitch := TRUE;

Mast1FlagsECU2PC.ECU2PC_TopPosition := MastControl.mastOben;

Mast1FlagsECU2PC.ECU2PC_BottomPosition := Mast1Height >= Mast1BottomPosition-1 AND Mast1Height <= Mast1BottomPosition+1;

Mast1FlagsECU2PC.ECU2PC_MovingUp := MastControl.aufbauen OR MastControl.mastAbsetzen;

Mast1FlagsECU2PC.ECU2PC_MovingDown := MastControl.abbauen;

Mast1FlagsECU2PC.ECU2PC_LocalUp := Inputs.TasteAusfahren;

Mast1FlagsECU2PC.ECU2PC_LocalDown := Inputs.TasteEinfahren;

Mast1FlagsECU2PC.ECU2PC_LimitSwitch4m := FALSE;

Mast1FlagsECU2PC.ECU2PC_LimitSwitchBottom := Inputs.EndschalterEingefahren;

Mast1FlagsECU2PC.ECU2PC_ParkPosition := Mast1FlagsECU2PC.ECU2PC_BottomPosition;

Mast1FlagsECU2PC.ECU2PC_MontagePos := NOT inputs.EndschalterAufgerichtet AND Mast1Height >= Mast1MontagePos-1 AND Mast1Height <= Mast1MontagePos+1;

Mast1MotorActiveTimeSeconds2 := Mast1MotorActiveTimeSeconds;
END_PROGRAM

(* POU Steuerung/PoweredByGenerator, ST *)
PROGRAM PoweredByGenerator
VAR_INPUT
	init: BOOL;
END_VAR
VAR
	rtTaste: R_TRIG;
	tofTaste: TOF;
END_VAR
IF init THEN
	(* Nach dem Einschalten erst mal aktivieren *)
	outputs.SchuetzGrundlast := TRUE;
END_IF

(* Taste entprellen *)
tofTaste(IN := inputs.TastePoweredByGenerator, PT := T#200ms);
rtTaste(CLK := tofTaste.Q);
IF rtTaste.Q THEN
	(* toggle *)
	outputs.SchuetzGrundlast := NOT outputs.SchuetzGrundlast;
END_IF
END_PROGRAM

(* POU Steuerung/MISC, ST *)
PROGRAM MISC
VAR
	TONInst: TON;
	OtherError: BOOL;
END_VAR
TONInst(IN := NOT TONInst.Q, PT:= T#500ms);
IF TONInst.Q THEN
	BlinkSlow := NOT BlinkSlow;
END_IF

IF NOT MasterPresent THEN
	FlagsPC2ECU := 0;
	Mast1FlagsPC2ECU := 0;
END_IF

Outputs.LEDAusgefahren := MastControl.mastOben;

Outputs.LEDEingefahren := Mast1FlagsECU2PC.ECU2PC_ParkPosition;

Outputs.LEDMontagePos := Mast1FlagsECU2PC.ECU2PC_MontagePos;

IntVoltage := SUPPLY_VOLTAGE_VBBS;

tasteAuf := inputs.TasteAusfahren OR Mast1FlagsPC2ECU.PC2ECU_MoveUp;
tasteAb := inputs.TasteEinfahren OR Mast1FlagsPC2ECU.PC2ECU_MoveDown;

IF tasteAuf AND tasteAb THEN
	tasteAuf := FALSE;
	tasteAb := FALSE;
END_IF
END_PROGRAM

(* POU InputsOutputs/WriteOutputs, FBD *)
PROGRAM WriteOutputs
VAR_INPUT
	OUT0: BOOL;
	OUT1: BOOL;
	OUT2: BOOL;
	OUT3: BOOL;
	OUT4: BOOL;
	OUT5: BOOL;
	OUT6: BOOL;
	OUT7: BOOL;
END_VAR
VAR
	_output: ARRAY[0..7] OF OUTPUT;
END_VAR
VAR CONSTANT
	ModeOutput_Off: BYTE := 0;
	ModeOutput_HighSide: BYTE := 2;
	ModeOutput_HighSide_Diag: BYTE := 15;
	ModeOutput_HighSide_Diag_Protection: BYTE := 16;
END_VAR
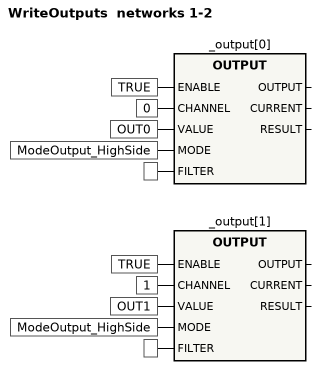
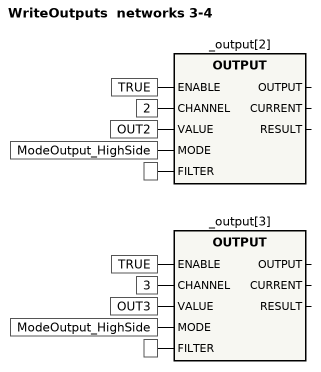
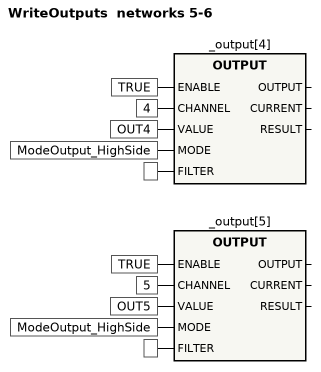
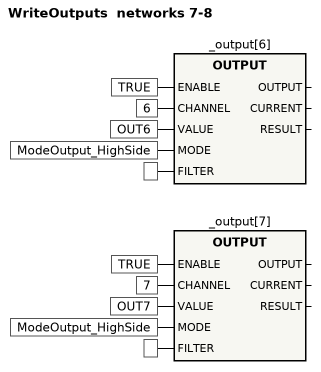
_FBD_ (* Function Block Diagram *)
NETWORK 1
	_output[0]:OUTPUT(ENABLE: TRUE, CHANNEL: 0, VALUE: OUT0, MODE: ModeOutput_HighSide, FILTER: )
NETWORK 2
	_output[1]:OUTPUT(ENABLE: TRUE, CHANNEL: 1, VALUE: OUT1, MODE: ModeOutput_HighSide, FILTER: )
NETWORK 3
	_output[2]:OUTPUT(ENABLE: TRUE, CHANNEL: 2, VALUE: OUT2, MODE: ModeOutput_HighSide, FILTER: )
NETWORK 4
	_output[3]:OUTPUT(ENABLE: TRUE, CHANNEL: 3, VALUE: OUT3, MODE: ModeOutput_HighSide, FILTER: )
NETWORK 5
	_output[4]:OUTPUT(ENABLE: TRUE, CHANNEL: 4, VALUE: OUT4, MODE: ModeOutput_HighSide, FILTER: )
NETWORK 6
	_output[5]:OUTPUT(ENABLE: TRUE, CHANNEL: 5, VALUE: OUT5, MODE: ModeOutput_HighSide, FILTER: )
NETWORK 7
	_output[6]:OUTPUT(ENABLE: TRUE, CHANNEL: 6, VALUE: OUT6, MODE: ModeOutput_HighSide, FILTER: )
NETWORK 8
	_output[7]:OUTPUT(ENABLE: TRUE, CHANNEL: 7, VALUE: OUT7, MODE: ModeOutput_HighSide, FILTER: )
_END_FBD_
END_PROGRAM
